TYPE DIOmodule:
STRUCT
	input	: ARRAY[0..7] OF BOOL;
	output	: ARRAY[0..7] OF BOOL;	
END_STRUCT
END_TYPE

(* stored: Version 1.1.0.1, ProductVersion 3.1.4024.11
   DUT DUT: Id {bdebea54-fa75-4aa3-ad60-6288b24cd565} *)
